// Mitsubishi GX Works2 project: servo1   PLC: Q03UDV

PROGRAM MAIN
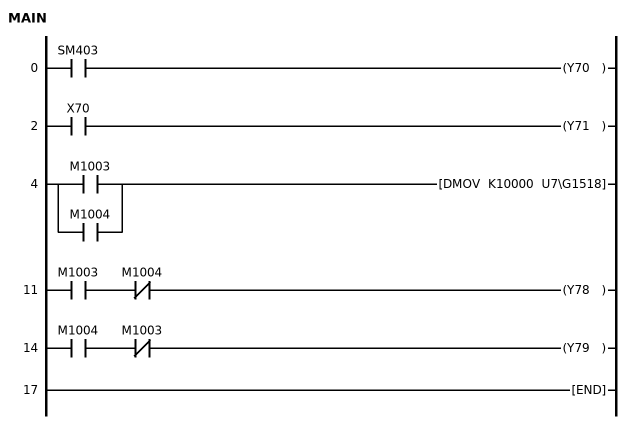
0     LD      SM403
      OUT     Y70
2     LD      X70
      OUT     Y71
4     LD      M1003
      OR      M1004
      DMOV    K10000 U7\G1518
11    LD      M1003
      ANI     M1004
      OUT     Y78
14    LD      M1004
      ANI     M1003
      OUT     Y79
17    END
END_PROGRAM
